FUNCTION F_LINT_ARG : ST_Arg
VAR_INPUT
	nInput : LINT;
END_VAR
VAR
	stArg : ST_Arg;
	sysVar_Info : __SYSTEM.VAR_INFO;
END_VAR

sysVar_Info 	:= __VARINFO(nInput);
stArg.TypeClass := sysVar_Info.TypeClass;
stArg.pValue 	:= 0;
stArg.diSize 	:= SIZEOF(nInput);
stArg.sValue 	:= TO_STRING(nInput); 
F_LINT_ARG := stArg;

END_FUNCTION

(* stored: Version 1.1.0.1, ProductVersion 3.1.4024.4
   POU F_LINT_ARG: Id {a37522cb-24e9-4b92-a610-944dc9c7b1d0}, SpecialFunc None *)
